PROGRAM Runner3
VAR
    foo : Foo;
    usesFoo : UsesFoo3(foo);
END_VAR

usesFoo();

END_PROGRAM

(* stored: Version 1.1.0.1, ProductVersion 3.1.4024.4
   POU Runner3: Id {e617f0e4-2b83-4d04-8109-40f7b1aee5ec}, SpecialFunc None *)
